FUNCTION_BLOCK itfActuateImplement IMPLEMENTS itfActuate
VAR_INPUT
END_VAR
VAR_OUTPUT
END_VAR
VAR
	Coil : BOOL;
	Start : BOOL;
	Stop : BOOL;
END_VAR

METHOD mTurnOffAuto : BOOL
pCoil := FALSE;
END_METHOD

METHOD mTurnOffManual : BOOL
IF pStop THEN
	pCoil := FALSE;
END_IF
END_METHOD

METHOD mTurnOnAuto : BOOL
pCoil := TRUE;
END_METHOD

METHOD mTurnOnManual : BOOL
IF pStart THEN
	pCoil := TRUE;
END_IF
END_METHOD

{warning 'add property implementation'}
PROPERTY pCoil : BOOL
GET
pCoil := Coil;
END_GET
SET
Coil := pCoil;
END_SET
END_PROPERTY

{warning 'add property implementation'}
PROPERTY pStart : BOOL
GET
pStart := Start;
END_GET
SET
Start := pStart;
END_SET
END_PROPERTY

{warning 'add property implementation'}
PROPERTY pStop : BOOL
GET
pStop := Stop;
END_GET
SET
Stop := pStop;
END_SET
END_PROPERTY

END_FUNCTION_BLOCK

(* stored: Version 1.1.0.1, ProductVersion 3.1.4024.12
   POU itfActuateImplement: Id {4d7328d8-3b44-4eaa-9d67-afb443720a15}, SpecialFunc None
   Method mTurnOffAuto: Id {087a05d9-5fcf-4297-8901-68efe5cafd20}
   Method mTurnOffManual: Id {ae7a5c7e-ea8e-45e0-a23a-e6cfff4cb6dc}
   Method mTurnOnAuto: Id {a45a887d-576a-4814-bca3-59e562303638}
   Method mTurnOnManual: Id {e3a9afca-1987-4adc-bc9c-5b4a3a284bd9}
   Property pCoil: Id {71dc4a1c-77f9-4779-8a10-3067f0bfdeb2}
   Get Get: Id {cf344ada-8149-4500-a4ce-70e5a59d4d98}
   Set Set: Id {92fa19e0-25fb-4d4d-a1ca-c2bfe4e65dd3}
   Property pStart: Id {96485657-947a-454e-9b9a-4d743bf29bd7}
   Get Get: Id {a8fd7b80-cdf8-417e-a7ed-e77ce1083422}
   Set Set: Id {8c6ec1a3-e800-49ea-ac50-f83ffb54f3cf}
   Property pStop: Id {92623c80-c715-454b-8df9-7f90e95cadc3}
   Get Get: Id {37994735-10c3-42a3-9bf8-cd68e1304c71}
   Set Set: Id {a7af93fc-9977-4c1f-93ed-e72e09528fd7} *)
